// TIA Portal V20 export
DATA_BLOCK "DB_UDI"   // DB30010
// stored: MemoryReserve 100, Namespace ProductionLine
   VAR
      ProductionLine : Struct
         Upstream : Struct
            Conveyor : Array[_.minProductionLine.._.maxProductionLine] of Bool;
         END_STRUCT;
         DownstreamAccu : Struct
            Stop : Struct
               Conveyor : Array[_.minProductionLine.._.maxProductionLine] of Bool;
            END_STRUCT;
         END_STRUCT;
         Interlock : Struct
            Stop : Struct
               Conveyor : Array[_.minProductionLine.._.maxProductionLine] of Bool;
            END_STRUCT;
         END_STRUCT;
         Fault : Struct
            Stop : Struct
               Conveyor : Array[_.minProductionLine.._.maxProductionLine] of Bool;
            END_STRUCT;
         END_STRUCT;
      END_STRUCT;
   END_VAR
BEGIN
   // ProductionLine.Upstream.Conveyor[1001] : A1.1.1
   // ProductionLine.Upstream.Conveyor[1002] : A1.1.2
   // ProductionLine.Upstream.Conveyor[1003] : A1.1.3
   // ProductionLine.Upstream.Conveyor[1004] : A1.1.4
   // ProductionLine.Upstream.Conveyor[1005] : A1.1.5
   // ProductionLine.Upstream.Conveyor[1006] : A1.1.6
   // ProductionLine.Upstream.Conveyor[1007] : A1.2.1
   // ProductionLine.Upstream.Conveyor[1008] : A1.2.2
   // ProductionLine.DownstreamAccu.Stop.Conveyor[1001] : A1.1.1
   // ProductionLine.DownstreamAccu.Stop.Conveyor[1002] : A1.1.2
   // ProductionLine.DownstreamAccu.Stop.Conveyor[1003] : A1.1.3
   // ProductionLine.DownstreamAccu.Stop.Conveyor[1004] : A1.1.4
   // ProductionLine.DownstreamAccu.Stop.Conveyor[1005] : A1.1.5
   // ProductionLine.DownstreamAccu.Stop.Conveyor[1006] : A1.1.6
   // ProductionLine.DownstreamAccu.Stop.Conveyor[1007] : A1.2.1
   // ProductionLine.DownstreamAccu.Stop.Conveyor[1008] : A1.2.2
   // ProductionLine.Interlock.Stop.Conveyor[1001] : A1.1.1
   // ProductionLine.Interlock.Stop.Conveyor[1002] : A1.1.2
   // ProductionLine.Interlock.Stop.Conveyor[1003] : A1.1.3
   // ProductionLine.Interlock.Stop.Conveyor[1004] : A1.1.4
   // ProductionLine.Interlock.Stop.Conveyor[1005] : A1.1.5
   // ProductionLine.Interlock.Stop.Conveyor[1006] : A1.1.6
   // ProductionLine.Interlock.Stop.Conveyor[1007] : A1.2.1
   // ProductionLine.Interlock.Stop.Conveyor[1008] : A1.2.2
   // ProductionLine.Fault.Stop.Conveyor[1001] : A1.1.1
   // ProductionLine.Fault.Stop.Conveyor[1002] : A1.1.2
   // ProductionLine.Fault.Stop.Conveyor[1003] : A1.1.3
   // ProductionLine.Fault.Stop.Conveyor[1004] : A1.1.4
   // ProductionLine.Fault.Stop.Conveyor[1005] : A1.1.5
   // ProductionLine.Fault.Stop.Conveyor[1006] : A1.1.6
   // ProductionLine.Fault.Stop.Conveyor[1007] : A1.2.1
   // ProductionLine.Fault.Stop.Conveyor[1008] : A1.2.2
END_DATA_BLOCK
